// Mitsubishi GX Works2 project: LRI   PLC: Q03UDV
// HELLOWORLD

PROGRAM MAIN
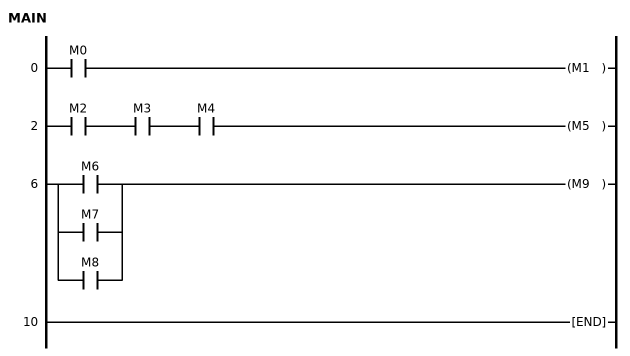
0     LD      M0
      OUT     M1
2     LD      M2
      AND     M3
      AND     M4
      OUT     M5
6     LD      M6
      OR      M7
      OR      M8
      OUT     M9
10    END
END_PROGRAM
